FUNCTION_BLOCK ASR2_TO_ASR (* Composite FB for convert bidirectional ASR2 to unidirectional ASR *)
  (* Standard: 61499-2; Function: ASR2_BIDIR forwards its incoming (EO_SET/EO_RESET) side out as plain unidirectional SET/RESET events via ASR_OUT. ASR_IN publishes SET/RESET onto the outgoing (EI_SET/EI_RESET) side of ASR2_BIDIR.; Description: Copyright (c) 2026 HR Agrartechnik GmbH This program and the accompanying materials are made available under the terms of the Eclipse Public License 2.0 which is available at https://www.eclipse.org/legal/epl-2.0/ SPDX-License-Identifier: EPL-2.0 *)
  (* Version 1.0, 2026-08-31, Franz Höpfinger, HR Agrartechnik GmbH, Initial Version *)
  PACKAGE adapter::conversion::bidirectional;
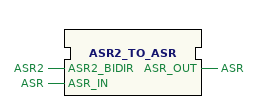
  SOCKETS
    ASR2_BIDIR : adapter::types::bidirectional::ASR2; (* Adapter Input: bidirectional tap, incoming side forwarded to ASR_OUT, outgoing side driven by ASR_IN *)
    ASR_IN : adapter::types::unidirectional::ASR; (* Adapter Input: unidirectional source *)
  END_SOCKETS
  PLUGS
    ASR_OUT : adapter::types::unidirectional::ASR; (* Adapter Output: mirrors ASR2_BIDIR's incoming (indication) side *)
  END_PLUGS
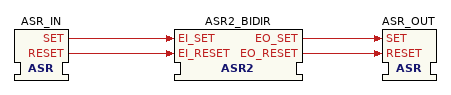
  EVENT_CONNECTIONS
    ASR2_BIDIR.EO_SET TO ASR_OUT.SET;
    ASR2_BIDIR.EO_RESET TO ASR_OUT.RESET;
    ASR_IN.SET TO ASR2_BIDIR.EI_SET;
    ASR_IN.RESET TO ASR2_BIDIR.EI_RESET;
  END_CONNECTIONS
END_FUNCTION_BLOCK
